{attribute 'qualified_only'}
VAR_GLOBAL
	Calibration_Pos_Moving			: 	BOOL	;
	HMI_Calibration_Pos_Move_PB		: 	BOOL	;
	Calibration_comp				: 	BOOL	;
	Calibration_OK					: 	BOOL	;
	All_Motor_Wait_Pos_Moving		: 	BOOL	;
	Calibration_Pos_Interlock 		: 	BOOL	;
	Data_Read_Comp					: 	BOOL	;
	Axis02_Data_Apply_Comp			: 	BOOL	;
	Axis03_Data_Apply_Comp			: 	BOOL	;
	Axis05_Data_Apply_Comp			: 	BOOL	;
END_VAR

(* stored: Version 1.1.0.1, ProductVersion 3.1.4024.15
   GVL GVL_Calibration_1: Id {2b4d4ec7-1f6a-48fa-9d05-6f75d9da2ee8} *)
